{attribute 'GeneratedUsingTerminal: EK1100-0000-0018'}
{attribute addProperty BoxType "EK1100-0000-0018"}
{attribute addProperty Id "Beckhoff_ELM3xxxEK1122Beckhoff_ELM3xxxEK1122_1A0BF0352A_0001_ELM3002_0000_0016ELM3002_3D4ED79F42A_0002_ELM3002_0000_0017ELM3002_3D4ED79F42A_0003_ELM3002_0000_0018ELM3002_3D4ED79F42A_0004_ELM3004_0000_0016ELM3004_177D76D464A_0005_ELM3004_0000_0017ELM3004_177D76D464A_0006_ELM3004_0000_0018ELM3004_177D76D464A_0007_ELM3004_0000_0019ELM3004_177D76D464"}
{attribute addProperty CRC "3967676929"}
{attribute addProperty Size "384"}
TYPE Beckhoff_ELM3xxx_EC7DF201 EXTENDS EK1100_1FC0878B :
STRUCT
	{attribute addProperty Name "Beckhoff_ELM3xxxEK1122"}
	{attribute addProperty PreviousPort "Beckhoff ELM3xxx : B"}
	Beckhoff_ELM3xxxEK1122 : Beckhoff_ELM3xxxEK1122_1A0BF035;
	{attribute addProperty Name "A_0001_ELM3002_0000_0016"}
	{attribute addProperty PreviousPort "Beckhoff ELM3xxxEK1122 : C"}
	A_0001_ELM3002_0000_0016 : ELM3002_3D4ED79F;
	{attribute addProperty Name "A_0002_ELM3002_0000_0017"}
	{attribute addProperty PreviousPort "A_0001(ELM3002-0000-0016) : B"}
	A_0002_ELM3002_0000_0017 : ELM3002_3D4ED79F;
	{attribute addProperty Name "A_0003_ELM3002_0000_0018"}
	{attribute addProperty PreviousPort "A_0002(ELM3002-0000-0017) : B"}
	A_0003_ELM3002_0000_0018 : ELM3002_3D4ED79F;
	{attribute addProperty Name "A_0004_ELM3004_0000_0016"}
	{attribute addProperty PreviousPort "A_0003(ELM3002-0000-0018) : B"}
	A_0004_ELM3004_0000_0016 : ELM3004_177D76D4;
	{attribute addProperty Name "A_0005_ELM3004_0000_0017"}
	{attribute addProperty PreviousPort "A_0004(ELM3004-0000-0016) : B"}
	A_0005_ELM3004_0000_0017 : ELM3004_177D76D4;
	{attribute addProperty Name "A_0006_ELM3004_0000_0018"}
	{attribute addProperty PreviousPort "A_0005(ELM3004-0000-0017) : B"}
	A_0006_ELM3004_0000_0018 : ELM3004_177D76D4;
	{attribute addProperty Name "A_0007_ELM3004_0000_0019"}
	{attribute addProperty PreviousPort "A_0006(ELM3004-0000-0018) : B"}
	A_0007_ELM3004_0000_0019 : ELM3004_177D76D4;
END_STRUCT
END_TYPE

(* stored: Version 1.2.0.0, ProductVersion 3.1.4024.9
   DUT Beckhoff_ELM3xxx_EC7DF201: Id {d1e4a00d-a614-4ff8-86b8-555f17f96693} *)
